FUNCTION_BLOCK {CATName} (* CAT Function Block Type *)
  (* Standard: 61499-2 *)
  (* Version 0.0, {MM/DD/YYYY}, {Author}, {YourOrg}, template *)
  PACKAGE {YourNamespace};
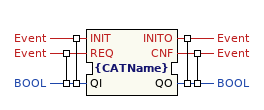
  EVENT_INPUT
    INIT WITH QI; (* Initialization Request *)
    REQ WITH QI; (* Normal Execution Request *)
  END_EVENT
  EVENT_OUTPUT
    INITO WITH QO; (* Initialization Confirm *)
    CNF WITH QO; (* Execution Confirmation *)
  END_EVENT
  VAR_INPUT
    QI : BOOL; (* Input event qualifier *)
  END_VAR
  VAR_OUTPUT
    QO : BOOL; (* Output event qualifier *)
  END_VAR
END_FUNCTION_BLOCK
